// TwinCAT 3 PLC project Untitled1
// ProgramVersion: 3.1.4026.1+972e9c44872ad038b353624a861fd7e3244e9f75
// libraries:
//   Tc2_EtherCAT, * (Beckhoff Automation GmbH)
//   Tc2_Standard, * (Beckhoff Automation GmbH)
//   Tc2_System, * (Beckhoff Automation GmbH)
// project tree:
//   / PlcTask.TcTTO
//   POUs/ MAIN.TcPOU
// real-time tasks:
//   TASK PlcTask: cycle T#10ms, priority 20, ADS port 350
// I/O:
//   DEVICE Device 1 (EtherCAT), AmsNetId 10.200.128.47.2.1
//     Term 1 (AX8620-0000-0105) [AX8620-0000-0105]
//       Drive 2 (AX8108-0200-0106) [AX8108-0200-0106 (1Ch. 8A servo axis, safe-motion)]
//         modules: Device, Device, Device, Device, Device, Device, Device, Device, Device, Device, Device (Safety), Device, Device, Device, Device, Device, Device, Device, Device, Device, Device, Device, Device, Device, Device, Device, Device, Device, Device, Device, Device, Ch A, Ch A, Ch A, Ch A, Ch A, Ch A, Ch A, Ch A, Ch A, Ch A, Ch A, Ch A, Ch A, Ch A, Ch A, Ch A, Ch A, Ch A, Ch A, Ch A, Ch A, Ch A, Ch A, Ch A, Ch A, Ch A

CONFIGURATION Untitled1
    RESOURCE PLC ON TwinCAT3
        TASK PlcTask(INTERVAL := T#10ms, PRIORITY := 20);
        PROGRAM MAIN WITH PlcTask : MAIN;
    END_RESOURCE
END_CONFIGURATION

// ---- POUs/MAIN.TcPOU
PROGRAM MAIN
VAR
	fbEcCoeSdoRead : FB_EcCoESdoRead;
	torque : REAL;
END_VAR

fbEcCoeSdoRead(
	sNetId:= '10.200.128.47.2.1', 
	nSlaveAddr:= 1002, 
	nSubIndex:=  17, 
	nIndex:= 16#32C0, 
	pDstBuf:= ADR(torque), 
	cbBufLen:= SIZEOF(torque), 
	bExecute:= , 
	);

END_PROGRAM
